(* CODESYS project Device.Plc Logic.Application.Area01.export

Project tree, tasks and I/O mapping:
  program Area01 [SFC]: Agitation_Cooling, Draining, Open_Control, RM_Fill
*)

// Area01
PROGRAM Area01
VAR
	Fill_Alowed: BOOL;
	Drain_Alowed:BOOL;
	VCU_101: VCU;//VCU of FV_101
	VCU_102: VCU; // Valv FV_102 VCU
	TimeOpen_101: TIME := T#11S250MS;
	TimeOpen_102: TIME := T#6S750MS;
	Flow_101: REAL :=2.67;
	Flow_102: REAL :=2.22;
	Flow_BA: REAL :=6.67;
	TimeOpen_BA: TIME := T#6S750MS;
	Delay_102: TON; // delay before FV_102 can be open
	
	// FV_102 TOF
	TOF_102: TOF;
	TON_102: TON;
	
	
	VCU_BA: VCU;
	
END_VAR
VAR // added by the converter: edge detectors and wires of the graphical bodies
    _ft1, _ft2 : F_TRIG;
END_VAR

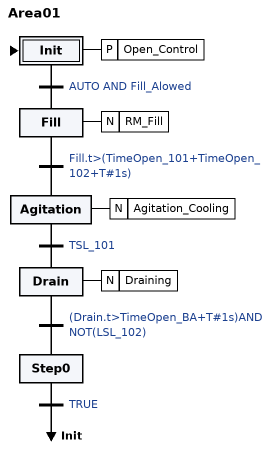
INITIAL_STEP Init:
    Open_Control(P);
END_STEP
TRANSITION FROM Init TO Fill
    := AUTO AND Fill_Alowed;
END_TRANSITION
STEP Fill:
    RM_Fill(N);
END_STEP
TRANSITION FROM Fill TO Agitation
    := Fill.t>(TimeOpen_101+TimeOpen_102+T#1s);
END_TRANSITION
STEP Agitation:
    Agitation_Cooling(N);
END_STEP
TRANSITION FROM Agitation TO Drain
    := TSL_101;
END_TRANSITION
STEP Drain:
    Draining(N);
END_STEP
TRANSITION FROM Drain TO Step0
    := (Drain.t>TimeOpen_BA+T#1s)AND NOT(LSL_102);
END_TRANSITION
STEP Step0:
END_STEP
TRANSITION FROM Step0 TO Init
    := TRUE;
END_TRANSITION

ACTION Agitation_Cooling:
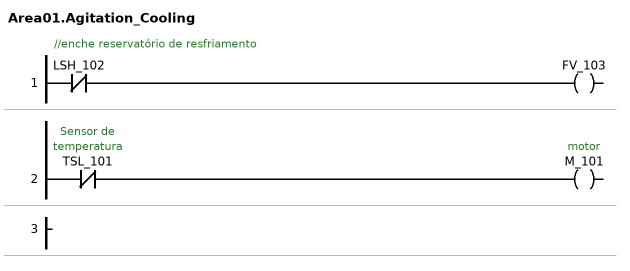
// NETWORK 1
// //enche reservatório de resfriamento
FV_103 := NOT LSH_102;

// NETWORK 2
//   TSL_101: Sensor de temperatura
//   M_101: motor
M_101 := NOT TSL_101;

// NETWORK 3
END_ACTION

ACTION Draining:
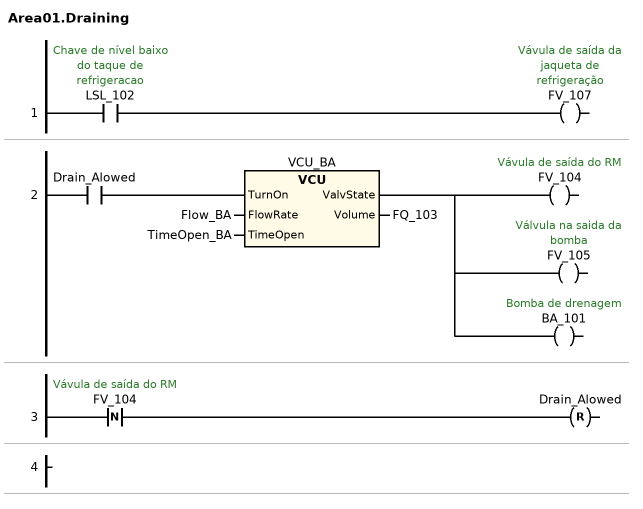
// NETWORK 1
//   LSL_102: Chave de nível baixo do taque de refrigeracao
//   FV_107: Vávula de saída da jaqueta de refrigeração
FV_107 := LSL_102;

// NETWORK 2
//   FQ_103: Totalizador Dry Martini
//   FV_104: Vávula de saída do RM
//   FV_105: Válvula na saida da bomba
//   BA_101: Bomba de drenagem
VCU_BA(TurnOn := Drain_Alowed, FlowRate := Flow_BA, TimeOpen := TimeOpen_BA, Volume => FQ_103); // VCU
FV_104 := VCU_BA.ValvState;
FV_105 := VCU_BA.ValvState;
BA_101 := VCU_BA.ValvState;

// NETWORK 3
//   FV_104: Vávula de saída do RM
_ft1(CLK := FV_104);
Drain_Alowed R= _ft1.Q;

// NETWORK 4
END_ACTION

ACTION Open_Control:
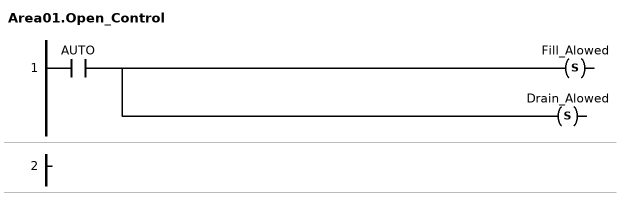
// NETWORK 1
Fill_Alowed S= AUTO;
Drain_Alowed S= AUTO;

// NETWORK 2
END_ACTION

ACTION RM_Fill:
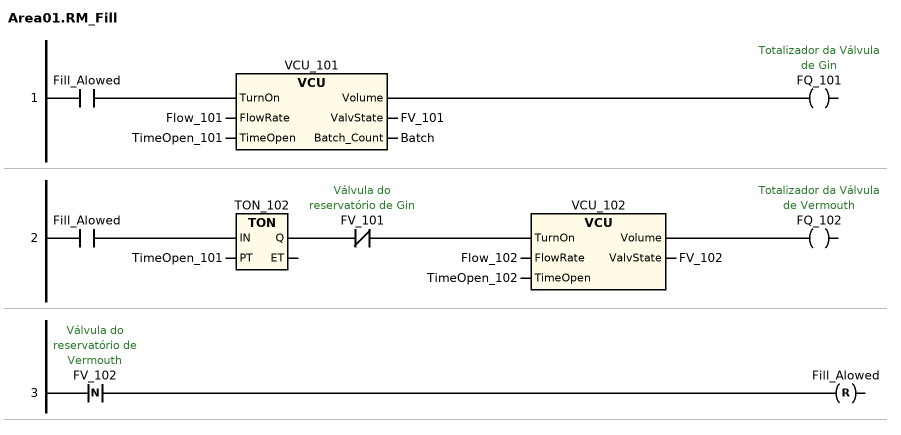
// NETWORK 1
//   VCU_101: VCU of FV_101
//   FV_101: Válvula do reservatório de Gin
//   FQ_101: Totalizador da Válvula de Gin
VCU_101(
    TurnOn := Fill_Alowed,
    FlowRate := Flow_101,
    TimeOpen := TimeOpen_101,
    ValvState => FV_101,
    Batch_Count => Batch); // VCU
FQ_101 := VCU_101.Volume;

// NETWORK 2
//   VCU_102: Valv FV_102 VCU
//   FV_101: Válvula do reservatório de Gin
//   FV_102: Válvula do reservatório de Vermouth
//   FQ_102: Totalizador da Válvula de Vermouth
TON_102(IN := Fill_Alowed, PT := TimeOpen_101); // TON
VCU_102(
    TurnOn := TON_102.Q AND NOT FV_101,
    FlowRate := Flow_102,
    TimeOpen := TimeOpen_102,
    ValvState => FV_102); // VCU
FQ_102 := VCU_102.Volume;

// NETWORK 3
//   FV_102: Válvula do reservatório de Vermouth
_ft2(CLK := FV_102);
Fill_Alowed R= _ft2.Q;
END_ACTION

END_PROGRAM
